FUNCTION_BLOCK RingCriticalSection (* Basic Function Block Type *)
  (* Standard: 61499-2 *)
  (* Version 0.2, 2003-12-04, JHC, Rockwell Automation, Renamed for better indexing. *)
  (* Version 0.1, 2002-11-05, JHC, Rockwell Automation, Corrected missing ST element in Algorithm REQ. *)
  (* Version 0.0, 2000-05-30, JHC, Rockwell Automation *)
  (* Compiler header: package fb.rt.cs725; *)
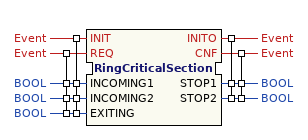
  EVENT_INPUT
    INIT WITH INCOMING1, INCOMING2, EXITING; (* Initialization Request *)
    REQ WITH INCOMING1, INCOMING2, EXITING; (* Normal Execution Request *)
  END_EVENT
  EVENT_OUTPUT
    INITO WITH STOP1, STOP2; (* Initialization Confirm *)
    CNF WITH STOP1, STOP2; (* Execution Confirmation *)
  END_EVENT
  VAR_INPUT
    INCOMING1 : BOOL; (* Input event qualifier *)
    INCOMING2 : BOOL;
    EXITING : BOOL;
  END_VAR
  VAR_OUTPUT
    STOP1 : BOOL; (* Output event qualifier *)
    STOP2 : BOOL;
  END_VAR
  VAR
    TOKEN_CLIENT : BOOL;
    TOKEN_BLOCK : BOOL;
  END_VAR
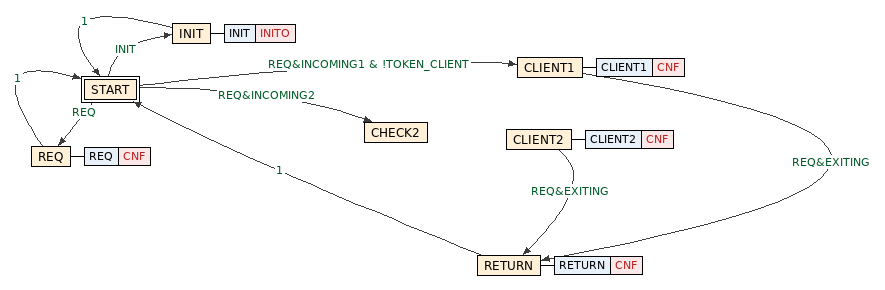
  EC_STATES
    START; (* Initial State *)
    INIT : INIT -> INITO; (* Initialization *)
    REQ : REQ -> CNF; (* Normal execution *)
    CLIENT1 : CLIENT1 -> CNF;
    CLIENT2 : CLIENT2 -> CNF;
    RETURN : RETURN -> CNF;
    CHECK2;
  END_STATES
  EC_TRANSITIONS
    START TO INIT := INIT;
    INIT TO START := 1;
    START TO REQ := REQ;
    REQ TO START := 1;
    CLIENT1 TO RETURN := REQ&EXITING;
    CLIENT2 TO RETURN := REQ&EXITING;
    RETURN TO START := 1;
    START TO CHECK2 := REQ&INCOMING2;
    START TO CLIENT1 := REQ&INCOMING1 & !TOKEN_CLIENT;
  END_TRANSITIONS
  ALGORITHM INIT IN ST: (* Initialization algorithm *)
TOKEN_BLOCK := FALSE;
TOKEN_CLIENT := FALSE;
  END_ALGORITHM
  ALGORITHM REQ IN ST: (* Normally executed algorithm *)
TOKEN_CLIENT := !TOKEN_CLIENT;
  END_ALGORITHM
  ALGORITHM CLIENT1 IN ST:
TOKEN_BLOCK := TRUE;
STOP1 := FALSE;
STOP2 := TRUE;
  END_ALGORITHM
  ALGORITHM CLIENT2 IN ST:
TOKEN_BLOCK := TRUE;
STOP1 := TRUE;
STOP2 := FALSE;
  END_ALGORITHM
  ALGORITHM RETURN IN ST:
TOKEN_BLOCK := FALSE;
STOP1 := FALSE;
STOP2 := FALSE;
  END_ALGORITHM
END_FUNCTION_BLOCK
